FUNCTION_BLOCK Section6
  (* Standard: 61499-2 *)
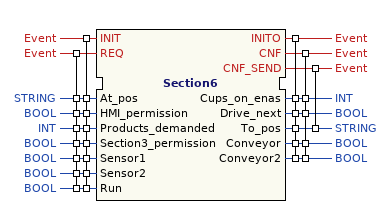
  EVENT_INPUT
    INIT WITH At_pos, HMI_permission, Products_demanded, Section3_permission, Sensor1, Sensor2, Run;
    REQ WITH At_pos, HMI_permission, Products_demanded, Section3_permission, Sensor1, Sensor2, Run;
  END_EVENT
  EVENT_OUTPUT
    INITO WITH Cups_on_enas, Drive_next, To_pos, Conveyor, Conveyor2;
    CNF WITH Cups_on_enas, Drive_next, Conveyor, Conveyor2;
    CNF_SEND WITH To_pos;
  END_EVENT
  VAR_INPUT
    At_pos : STRING;
    HMI_permission : BOOL;
    Products_demanded : INT;
    Section3_permission : BOOL;
    Sensor1 : BOOL;
    Sensor2 : BOOL;
    Run : BOOL;
  END_VAR
  VAR_OUTPUT
    Cups_on_enas : INT;
    Drive_next : BOOL;
    To_pos : STRING;
    Conveyor : BOOL;
    Conveyor2 : BOOL;
  END_VAR
  FBS
    FB2 : DisableConveyor;
    FB3 : DisableConveyor;
    FB1 : Section6Ctrl;
    FB4 : E_MERGE;
  END_FBS
  EVENT_CONNECTIONS
    INIT TO FB1.INIT;
    FB1.CNF TO FB2.REQ;
    REQ TO FB2.REQ;
    FB1.INITO TO FB2.INIT;
    FB2.CNF TO FB4.EI1;
    REQ TO FB1.REQ;
    FB1.CNF_SEND TO CNF_SEND;
    FB1.INITO TO FB3.INIT;
    REQ TO FB3.REQ;
    FB1.CNF TO FB3.REQ;
    FB3.CNF TO FB4.EI2;
    FB4.EO TO CNF;
  END_CONNECTIONS
  DATA_CONNECTIONS
    Run TO FB2.QI;
    FB1.Conveyor TO FB2.ConvIn;
    FB2.ConvOut TO Conveyor;
    Sensor2 TO FB1.Sensor2;
    Sensor1 TO FB1.Sensor1;
    Products_demanded TO FB1.Product_demanded;
    HMI_permission TO FB1.HMI_permission;
    At_pos TO FB1.At_pos;
    Section3_permission TO FB1.Section3_permission;
    FB1.To_pos TO To_pos;
    FB1.Drive_next TO Drive_next;
    FB1.Cups_on_enas TO Cups_on_enas;
    Run TO FB3.QI;
    FB1.Conveyor2 TO FB3.ConvIn;
    FB3.ConvOut TO Conveyor2;
  END_CONNECTIONS
END_FUNCTION_BLOCK
